// TwinCAT 3 PLC project PLC
// ProgramVersion: 3.1.4024.0
// libraries:
//   EfficientIO Communicator, * (EfficientIO)
//   Lynus Persistent Data V1, * (Lynus AG)
//   Lynus Standards, * (Lynus AG)
//   Tc2_ModbusRTU, * (Beckhoff Automation GmbH)
//   Tc2_SerialCom, * (Beckhoff Automation GmbH)
//   Tc2_Standard, * (Beckhoff Automation GmbH)
//   Tc2_System, * (Beckhoff Automation GmbH)
//   Tc2_Utilities, * (Beckhoff Automation GmbH)
//   Tc3_Module, * (Beckhoff Automation GmbH)
// project tree:
//   DUTs/ ModbusRTURequest.TcDUT
//   / FastTask.TcTTO, MiddleTask.TcTTO, SlowTask.TcTTO
//   FB/ FB_ModBus_2Registers_FC4_T.TcPOU (not stored), F_Convert_Reg_to_Real.TcPOU (not stored), MODBUS_RTU_EcoForest.TcPOU, MODBUS_RTU_Vallox.TcPOU
//   POUs/ prgCom.TcPOU, prgHeatPump.TcPOU, prgMiddle.TcPOU, prgPD.TcPOU, prgRoomVentilaton.TcPOU, prgVar.TcPOU
// real-time tasks:
//   TASK FastTask: cycle T#5ms, priority 19, ADS port 351
//   TASK MiddleTask: cycle T#10ms, priority 20, ADS port 352
//   TASK SlowTask: cycle T#20ms, priority 21, ADS port 353
// I/O:
//   DEVICE Gerät 2 (CX-BK)
//     Box 1 (CX-BK)
// variable links:
//   PLC/PLC Instance <-> Device 2 (CX-BK)/Box 1 (CX-BK)
//     MiddleTask Inputs/MODBUS_RTU_EcoForest.fbModbusRtuMaster_KL6x22B.InData/D[{0..21}] <-> Term 2 (KL6041)/Channel 1/Data In {0..21}  (22 links)
//     MiddleTask Inputs/MODBUS_RTU_EcoForest.fbModbusRtuMaster_KL6x22B.InData/Status <-> Term 2 (KL6041)/Channel 1/Status
//     MiddleTask Inputs/MODBUS_RTU_Vallox.fbModbusRtuMaster_KL6x22B.InData/D[{0..21}] <-> Term 3 (KL6041)/Channel 1/Data In {0..21}  (22 links)
//     MiddleTask Inputs/MODBUS_RTU_Vallox.fbModbusRtuMaster_KL6x22B.InData/Status <-> Term 3 (KL6041)/Channel 1/Status
//     MiddleTask Outputs/MODBUS_RTU_EcoForest.fbModbusRtuMaster_KL6x22B.OutData/Ctrl <-> Term 2 (KL6041)/Channel 1/Ctrl
//     MiddleTask Outputs/MODBUS_RTU_EcoForest.fbModbusRtuMaster_KL6x22B.OutData/D[{0..21}] <-> Term 2 (KL6041)/Channel 1/Data Out {0..21}  (22 links)
//     MiddleTask Outputs/MODBUS_RTU_Vallox.fbModbusRtuMaster_KL6x22B.OutData/Ctrl <-> Term 3 (KL6041)/Channel 1/Ctrl
//     MiddleTask Outputs/MODBUS_RTU_Vallox.fbModbusRtuMaster_KL6x22B.OutData/D[{0..21}] <-> Term 3 (KL6041)/Channel 1/Data Out {0..21}  (22 links)
//     SlowTask Inputs/prgMiddle.uint_State <-> Inputs/State

CONFIGURATION PLC
    RESOURCE PLC ON TwinCAT3
        TASK FastTask(INTERVAL := T#5ms, PRIORITY := 19);
        TASK MiddleTask(INTERVAL := T#10ms, PRIORITY := 20);
        TASK SlowTask(INTERVAL := T#20ms, PRIORITY := 21);
        PROGRAM prgPD WITH FastTask : prgPD;
        PROGRAM prgVar WITH FastTask : prgVar;
        PROGRAM prgMiddle WITH MiddleTask : prgMiddle;
        PROGRAM prgCom WITH SlowTask : prgCom;
    END_RESOURCE
END_CONFIGURATION

// ---- DUTs/ModbusRTURequest.TcDUT
TYPE ModbusRTURequest :
STRUCT
	byteClientSlaveID	:BYTE;
	uintStartAddress	:UINT;
	uintNoOfWords		:UINT;
	mError				:BOOL;
	udintErrorID		:MODBUS_ERRORS;
	udintBytesReceived	:UDINT;
	timerErrorTimer		:TON;
	timerOKTimer		:TON;
	wArrayReceiveBuffer	:ARRAY[0..130] OF WORD;
	udintReceiveBufferAddress	:UDINT;
	strErrorMessage		:STRING(50);
	udintCommErrorCounter		:UDINT;
	udintCommSuccessCounter		:UDINT;
	timeTimeForRequest	:TIME;
	mRequestActive		:BOOL;
	intDeviceClass		:INT;
	intDeviceNumber		:INT;
END_STRUCT
END_TYPE

// ---- POUs/prgPD.TcPOU
PROGRAM prgPD
VAR
	fbPers						: FB_WritePersistentData_General;
	fb_Reboot		: NT_reboot;
	m_Reboot		: BOOL:=FALSE;
END_VAR

fbPers(
	eSaveModeData:= eUSVSaveMode.eSaveEventBased, 
	bLoadPersistentDataOk=> , 
	bError=> , 
	bySaveProcess=> , 
	dwStorageLast24h=> , 
	udiErrorCode=> );
	
	
fb_Reboot(	netid := '',
			delay := 2,
			start := m_Reboot);

END_PROGRAM

// ---- POUs/prgVar.TcPOU
PROGRAM prgVar
VAR
	fbVar			: FB_VarInfo_V3;
	fbrw1			: FB_ReadWrite_V2;
END_VAR

fbVar(
	bReadInfo:= , 
	eTMCFile:= eSelectTMCFile.eDontUseTMCFile, 
	eSavePositionTMCFile:= eSavePositionOnPLC.ePostionHardDisk, 
	udiCounterFoundVariables=> , 
	bError=> , 
	bBusy=> , 
	byProgress=> , 
	udiErrorCodeOut=> , 
	eErrorVarInfo_Out=> , 
	sVarWithError=> );
fbVar();
fbVar();
	
fbRW1(	eUploadType := eSelectDataUploadType.e_Change_Intervall5min,
		bBusy=> , 
		bError=> , 
		udiErrorCodeOut=> , 
		eErrorReadWrite_Out=> );

END_PROGRAM

// ---- POUs/prgMiddle.TcPOU
PROGRAM prgMiddle
VAR
	i: INT;
	int_LiveCount_5min:INT;								//{#lynus.ag#()}
	ton_5min: Ton;
	uint_State								AT%I* 	: UINT;		//{#lynus.ag#()}
	mtest: BOOL;

END_VAR

i:= i+1;
ton_5min( 	In := NOT ton_5min.Q,
			PT := T#5M);
IF ton_5min.Q THEN
	int_LiveCount_5min := int_LiveCount_5min+1;
END_IF

prgHeatPump();
prgRoomVentilaton();

END_PROGRAM

// ---- POUs/prgHeatPump.TcPOU
PROGRAM prgHeatPump
VAR
	fb_word_to_float	:FB_CV_WORD_TO_REAL_FLOAT;
	real_ProductionTemperatureOut		: REAL;									//{#lynus.ag#()}
	real_ProductionTemperatureIn		: REAL;									//{#lynus.ag#()}
	real_CompresorSuctionPressure		: REAL;									//{#lynus.ag#()}
	real_CompressorDischargePressure	: REAL;									//{#lynus.ag#()}
	real_DHWTemperature					: REAL;									//{#lynus.ag#()}
	real_OutdoorTemperature				: REAL;									//{#lynus.ag#()}
	real_BrineCircuitPressure			: REAL;									//{#lynus.ag#()}
	real_ProductionCircuitPressure		: REAL;									//{#lynus.ag#()}
	real_CompressorStartTempForDHW		: REAL;									//{#lynus.ag#()}
	real_COP							: REAL;									//{#lynus.ag#()}
	real_PF								: REAL;									//{#lynus.ag#()}
	real_CondensationTemperature		: REAL;									//{#lynus.ag#()}
	real_Superheat						: REAL;									//{#lynus.ag#()}
	real_ExpansionValvePosition			: REAL;									//{#lynus.ag#()}
	real_SetpointDHWBUS					: REAL;									//{#lynus.ag#()}
	real_BUSHeatingDG1Setpoint			: REAL;									//{#lynus.ag#()}
	real_BUSHeatingSG2Setpoint			: REAL;									//{#lynus.ag#()}
	real_BUSHeatingSG3Setpoint			: REAL;									//{#lynus.ag#()}
	real_BUSHeatingSG4Setpoint			: REAL;									//{#lynus.ag#()}
	real_BUSCoolingDG1Setpoint			: REAL;									//{#lynus.ag#()}
	real_BUSCoolingSG2Setpoint			: REAL;									//{#lynus.ag#()}
	real_BUSCoolingSG3Setpoint			: REAL;									//{#lynus.ag#()}
	real_BUSCoolingSG4Setpoint			: REAL;									//{#lynus.ag#()}
	real_SupplytemperatureSG2			: REAL;									//{#lynus.ag#()}
	real_SupplytemperatureSG3			: REAL;									//{#lynus.ag#()}
	real_SupplytemperatureSG4			: REAL;									//{#lynus.ag#()}
	real_DHWStarttemperature			: REAL;									//{#lynus.ag#()}
	real_Evaporationtemperature			: REAL;									//{#lynus.ag#()}
	real_Heatingbuffertanktemp			: REAL;									//{#lynus.ag#()}
	real_Coolingbuffertanktemp			: REAL;									//{#lynus.ag#()}
	real_EER							: REAL;									//{#lynus.ag#()}
	real_Compresordischargetemp			: REAL;									//{#lynus.ag#()}
	real_Surplusactivationsetpoint		: REAL;									//{#lynus.ag#()}
	real_Consumptionlimitsetpoint 		: REAL;									//{#lynus.ag#()}
	real_CompressorRPM					: REAL;									//{#lynus.ag#()}
	real_ScrollTemp						: REAL;									//{#lynus.ag#()}
	real_Invertertemperature			: REAL;									//{#lynus.ag#()}
	real_Powerconsumption				: REAL;									//{#lynus.ag#()}
	real_Condensationcapacity			: REAL;									//{#lynus.ag#()}

	real_Heatpumpstate					: REAL;									//{#lynus.ag#()}
	// 1=Off; 2=On; 3=Emergency; 0=Keyboard
	real_Workingprogram					: REAL;									//{#lynus.ag#()}
	// 1=Winter;2=Summer; 3=Mixed; 0=Keyboard
	real_BUS_DHWDemand					: REAL;									//{#lynus.ag#()}
	real_BUS_SG2Demand					: REAL;									//{#lynus.ag#()}
	real_BUS_SG3Demand					: REAL;									//{#lynus.ag#()}
	real_BUS_SG4Demand					: REAL;									//{#lynus.ag#()}
//	real_			: REAL;									//{#lynus.ag#()}
//	real_			: REAL;									//{#lynus.ag#()}
	
	bool_HP_Alarm					: BOOL;								//{#lynus.ag#()}
	bool_HP_BusControlEnable		: BOOL;								//{#lynus.ag#()}

	mTest: BOOL;

END_VAR

MODBUS_RTU_EcoForest();
IF MODBUS_RTU_EcoForest.structArrayModbusRTU[1].wArrayReceiveBuffer[10]<>0 THEN 	
	real_ProductionTemperatureOut 	:=INT_TO_REAL(WORD_TO_INT(MODBUS_RTU_EcoForest.structArrayModbusRTU[1].wArrayReceiveBuffer[2]))/10;
	real_ProductionTemperatureIn 	:=INT_TO_REAL(WORD_TO_INT(MODBUS_RTU_EcoForest.structArrayModbusRTU[1].wArrayReceiveBuffer[3]))/10;
	real_CompresorSuctionPressure 	:=INT_TO_REAL(WORD_TO_INT(MODBUS_RTU_EcoForest.structArrayModbusRTU[1].wArrayReceiveBuffer[5]))/10;
	real_CompressorDischargePressure:=int_to_real(word_to_int(MODBUS_RTU_EcoForest.structArrayModbusRTU[1].wArrayReceiveBuffer[6]))/10;
	real_DHWTemperature				:=int_to_real(word_to_int(MODBUS_RTU_EcoForest.structArrayModbusRTU[1].wArrayReceiveBuffer[7]))/10;
	real_OutdoorTemperature			:=int_to_real(word_to_int(MODBUS_RTU_EcoForest.structArrayModbusRTU[1].wArrayReceiveBuffer[10]))/10;
	real_BrineCircuitPressure		:=int_to_real(word_to_int(MODBUS_RTU_EcoForest.structArrayModbusRTU[1].wArrayReceiveBuffer[12]))/10;
	real_ProductionCircuitPressure	:=int_to_real(word_to_int(MODBUS_RTU_EcoForest.structArrayModbusRTU[1].wArrayReceiveBuffer[13]))/10;
	real_CompressorStartTempForDHW	:=int_to_real(word_to_int(MODBUS_RTU_EcoForest.structArrayModbusRTU[1].wArrayReceiveBuffer[14]))/10;
END_IF
IF (MODBUS_RTU_EcoForest.structArrayModbusRTU[2].wArrayReceiveBuffer[7])/10 <> 0 THEN	
	real_COP						:= INT_TO_REAL(WORD_TO_INT(MODBUS_RTU_EcoForest.structArrayModbusRTU[2].wArrayReceiveBuffer[7]))/10;	
	real_PF							:= INT_TO_REAL(WORD_TO_INT(MODBUS_RTU_EcoForest.structArrayModbusRTU[2].wArrayReceiveBuffer[8]))/10;
END_IF	
IF  (MODBUS_RTU_EcoForest.structArrayModbusRTU[3].wArrayReceiveBuffer[0])/10 <>0 THEN 	
	real_CondensationTemperature	:= INT_TO_REAL(WORD_TO_INT(MODBUS_RTU_EcoForest.structArrayModbusRTU[3].wArrayReceiveBuffer[0]))/10;	
END_IF	
IF (MODBUS_RTU_EcoForest.structArrayModbusRTU[4].wArrayReceiveBuffer[1])/10 <> 0 THEN
	real_Superheat					:= INT_TO_REAL(WORD_TO_INT(MODBUS_RTU_EcoForest.structArrayModbusRTU[4].wArrayReceiveBuffer[0]))/10;	
	real_ExpansionValvePosition		:= int_to_real(word_to_int(MODBUS_RTU_EcoForest.structArrayModbusRTU[4].wArrayReceiveBuffer[1]))/10;	
	real_SetpointDHWBUS				:= int_to_real(word_to_int(MODBUS_RTU_EcoForest.structArrayModbusRTU[4].wArrayReceiveBuffer[2]))/10;	
	real_BUSHeatingDG1Setpoint		:= int_to_real(word_to_int(MODBUS_RTU_EcoForest.structArrayModbusRTU[4].wArrayReceiveBuffer[3]))/10;	
	real_BUSHeatingSG2Setpoint		:= int_to_real(word_to_int(MODBUS_RTU_EcoForest.structArrayModbusRTU[4].wArrayReceiveBuffer[4]))/10;	
	real_BUSHeatingSG3Setpoint		:= int_to_real(word_to_int(MODBUS_RTU_EcoForest.structArrayModbusRTU[4].wArrayReceiveBuffer[5]))/10;	
	real_BUSHeatingSG4Setpoint		:= int_to_real(word_to_int(MODBUS_RTU_EcoForest.structArrayModbusRTU[4].wArrayReceiveBuffer[6]))/10;	
	real_BUSCoolingDG1Setpoint		:= int_to_real(word_to_int(MODBUS_RTU_EcoForest.structArrayModbusRTU[4].wArrayReceiveBuffer[7]))/10;	
	real_BUSCoolingSG2Setpoint		:= int_to_real(word_to_int(MODBUS_RTU_EcoForest.structArrayModbusRTU[4].wArrayReceiveBuffer[8]))/10;	
	real_BUSCoolingSG3Setpoint		:= int_to_real(word_to_int(MODBUS_RTU_EcoForest.structArrayModbusRTU[4].wArrayReceiveBuffer[9]))/10;	
	real_BUSCoolingSG4Setpoint		:= INT_TO_REAL(WORD_TO_INT(MODBUS_RTU_EcoForest.structArrayModbusRTU[4].wArrayReceiveBuffer[10]))/10;	
END_IF


IF (MODBUS_RTU_EcoForest.structArrayModbusRTU[7].wArrayReceiveBuffer[1])/10 <> 0 THEN 
	real_SupplytemperatureSG2		:= INT_TO_REAL(WORD_TO_INT(MODBUS_RTU_EcoForest.structArrayModbusRTU[7].wArrayReceiveBuffer[0]))/10;	
	real_SupplytemperatureSG3		:= int_to_real(word_to_int(MODBUS_RTU_EcoForest.structArrayModbusRTU[7].wArrayReceiveBuffer[1]))/10;	
	real_SupplytemperatureSG4		:= int_to_real(word_to_int(MODBUS_RTU_EcoForest.structArrayModbusRTU[7].wArrayReceiveBuffer[2]))/10;	
	real_DHWStarttemperature		:= int_to_real(word_to_int(MODBUS_RTU_EcoForest.structArrayModbusRTU[7].wArrayReceiveBuffer[3]))/10;	
	real_Evaporationtemperature		:= int_to_real(word_to_int(MODBUS_RTU_EcoForest.structArrayModbusRTU[7].wArrayReceiveBuffer[4]))/10;	
	real_Heatingbuffertanktemp		:= int_to_real(word_to_int(MODBUS_RTU_EcoForest.structArrayModbusRTU[7].wArrayReceiveBuffer[5]))/10;	
	real_Coolingbuffertanktemp		:= int_to_real(word_to_int(MODBUS_RTU_EcoForest.structArrayModbusRTU[7].wArrayReceiveBuffer[6]))/10;	
	real_EER						:= int_to_real(word_to_int(MODBUS_RTU_EcoForest.structArrayModbusRTU[7].wArrayReceiveBuffer[7]))/10;	
	real_Compresordischargetemp		:= int_to_real(word_to_int(MODBUS_RTU_EcoForest.structArrayModbusRTU[7].wArrayReceiveBuffer[8]))/10;	
END_IF

IF (MODBUS_RTU_EcoForest.structArrayModbusRTU[8].wArrayReceiveBuffer[0])/10 <> 0 THEN
	real_Surplusactivationsetpoint	:= INT_TO_REAL(WORD_TO_INT(MODBUS_RTU_EcoForest.structArrayModbusRTU[8].wArrayReceiveBuffer[0]))/10;	
	real_Consumptionlimitsetpoint	:= INT_TO_REAL(WORD_TO_INT(MODBUS_RTU_EcoForest.structArrayModbusRTU[8].wArrayReceiveBuffer[1]))/10;	
END_IF

IF MODBUS_RTU_EcoForest.structArrayModbusRTU[5].wArrayReceiveBuffer[3] <> 0 THEN		
	real_CompressorRPM 				:= INT_TO_REAL(WORD_TO_INT(MODBUS_RTU_EcoForest.structArrayModbusRTU[5].wArrayReceiveBuffer[0]));
	real_ScrollTemp					:= int_to_real(word_to_int(MODBUS_RTU_EcoForest.structArrayModbusRTU[5].wArrayReceiveBuffer[2]));
	real_Invertertemperature		:= int_to_real(word_to_int(MODBUS_RTU_EcoForest.structArrayModbusRTU[5].wArrayReceiveBuffer[3]));
END_IF

IF MODBUS_RTU_EcoForest.structArrayModbusRTU[6].wArrayReceiveBuffer[3] <> 0 THEN
	real_Powerconsumption			:= INT_TO_REAL(WORD_TO_INT(MODBUS_RTU_EcoForest.structArrayModbusRTU[6].wArrayReceiveBuffer[2]));		
	real_Condensationcapacity		:= INT_TO_REAL(WORD_TO_INT(MODBUS_RTU_EcoForest.structArrayModbusRTU[6].wArrayReceiveBuffer[3]));		
END_IF

IF MODBUS_RTU_EcoForest.structArrayModbusRTU[9].wArrayReceiveBuffer[8] <> 0 THEN // [8] = Start counter
	real_Heatpumpstate		:= INT_TO_REAL(WORD_TO_INT(MODBUS_RTU_EcoForest.structArrayModbusRTU[9].wArrayReceiveBuffer[0]));	
	real_Workingprogram		:= INT_TO_REAL(WORD_TO_INT(MODBUS_RTU_EcoForest.structArrayModbusRTU[9].wArrayReceiveBuffer[1]));	
	real_BUS_DHWDemand		:= INT_TO_REAL(WORD_TO_INT(MODBUS_RTU_EcoForest.structArrayModbusRTU[9].wArrayReceiveBuffer[2]));
	real_BUS_SG2Demand		:= INT_TO_REAL(WORD_TO_INT(MODBUS_RTU_EcoForest.structArrayModbusRTU[9].wArrayReceiveBuffer[4]));	
	real_BUS_SG3Demand		:= INT_TO_REAL(WORD_TO_INT(MODBUS_RTU_EcoForest.structArrayModbusRTU[9].wArrayReceiveBuffer[5]));	
	real_BUS_SG4Demand		:= INT_TO_REAL(WORD_TO_INT(MODBUS_RTU_EcoForest.structArrayModbusRTU[9].wArrayReceiveBuffer[6]));	
END_IF
	

bool_HP_Alarm 				:= WORD_TO_BOOL(MODBUS_RTU_EcoForest.structArrayModbusRTU[10].wArrayReceiveBuffer[0]);
bool_HP_BusControlEnable	:= WORD_TO_BOOL(MODBUS_RTU_EcoForest.structArrayModbusRTU[10].wArrayReceiveBuffer[3]);

//			:= INT_TO_REAL(WORD_TO_INT(MODBUS_RTU_EcoForest.structArrayModbusRTU[].wArrayReceiveBuffer[]));	
//			:= INT_TO_REAL(WORD_TO_INT(MODBUS_RTU_EcoForest.structArrayModbusRTU[].wArrayReceiveBuffer[]));

END_PROGRAM

// ---- FB/MODBUS_RTU_EcoForest.TcPOU
PROGRAM MODBUS_RTU_EcoForest

VAR_INPUT

END_VAR
VAR_OUTPUT
	dword_MB_Error		:ARRAY[1..3] OF DWORD;
END_VAR
VAR
//	fbModbusRtuMaster_KL6x22B: ModbusRtuMaster_KL6x22B;
	fbModbusRtuMaster_KL6x22B: ModbusRtuMasterV2_KL6x22B;
	fbConfigKL6041 : KL6Configuration;
	uintPollOrderCount: UINT;
	mBusy: BOOL;
	mError: BOOL;
	mStart: BOOL;
	udintMemoryDestAddress: UDINT;
	udintBytesReceived: UDINT;
	intState: INT:=0;
	timerT1: TON;
	timeWaitT1: TIME:=T#500MS;
	timeWaitT2: TIME:=T#500MS;
	timeNoRxTimeout:	TIME:=T#2S;
	timerT2: TON;

	fb_F_TRIG1: F_TRIG;
	timerTimeout: TON;
	mError_Rx: BOOL;
	udintErrorID: MODBUS_ERRORS;
	byteClientSlaveID: BYTE;
	uintNoOfWords: UINT;
	uintStartAddress: UINT;
	dw_Mask: DWORD;
	dw_Mask_Not: DWORD;
	uint_TestPollOrder: UINT;
	mTestMode: BOOL;
	mInit_Done: BOOL;
	
	structArrayModbusRTU	:ARRAY[1..60] OF ModbusRTURequest;
	uintMaxModbusRTUOrders: UINT;
	mExecute: BOOL;
	int_Handshake: ComHandshake_t:=4;
	mode: ComSerialLineMode_t:=3;
	byte_DataBits: BYTE:=8;
	Word_Quantity: WORD;
	Word_Adress: WORD;
	uint_Length: UINT;
	udint_Write_Value:UDINT;
	udintMemoryDestAddress_Write: POINTER TO UDINT;
	mStartWrite: BOOL;
	i:uint;
END_VAR

(*
The function block "ModbusRtuMaster_KL6x22B" has 22 bytes where it communicates with the plc
software. These 22 bytes have to be assigned to the hardware device (for example KL/EL6021) in the
system manager plus the control and status byte.
If devices with less then 22 bytes are used, the other function blocks have to be used (for 5 bytes for example).
*)

(*
IF fbModbusRtuMaster_KL6x22B.MBmaster.TimeoutTON.Q=TRUE AND mTimeOUT_Qold=FALSE THEN mTimeOUT_Q_Rising; END_IF
mTimeOUT_Qold:=fbModbusRtuMaster_KL6x22B.MBmaster.TimeoutTON.Q;
*)

fb_F_TRIG1(CLK:=mBusy);

CASE intState OF

0: 	(* reset the start bit *)
	mStart:=FALSE;
	IF mInit_Done AND NOT fbConfigKL6041.Busy THEN 
		intState:=10;
		mExecute:=FALSE;		
	ELSE
		INIT();
		mExecute:=TRUE;		// necessary to write the communication parameters to the KL terminal. only necessary once if the terminal is brand new
	END_IF
10:
	(* set next poll order *)
	uintPollOrderCount:=uintPollOrderCount+1; (* next slave *)
	WHILE NOT structArrayModbusRTU[uintPollOrderCount].mRequestActive DO
		uintPollOrderCount:=uintPollOrderCount+1; (* next slave *)
	END_WHILE
	
	(* trouble shooting *)
	IF mTestMode THEN
		uintPollOrderCount:=uint_TestPollOrder; (* next slave *)
	END_IF
	
	IF uintPollOrderCount > uintMaxModbusRTUOrders OR uintPollOrderCount<1 THEN
		uintPollOrderCount:=1;
	END_IF

	udintMemoryDestAddress:=ADR(structArrayModbusRTU[uintPollOrderCount].wArrayReceiveBuffer[0]);
	structArrayModbusRTU[uintPollOrderCount].udintBytesReceived:=0;
	mStart:=TRUE;
	timerTimeout.IN:=TRUE;
	intState:=20;

20: (* wait for busy falling or time out *)
	IF fb_F_TRIG1.Q OR timerTimeout.Q THEN

		(* check answer time *)
		structArrayModbusRTU[uintPollOrderCount].timeTimeForRequest:=timerTimeout.ET;

		(* reset timer *)
		timerTimeout.IN:=FALSE;

		(* reset start bit *)
		mStart:=FALSE;

		(* save number of bytes received *)
		structArrayModbusRTU[uintPollOrderCount].udintBytesReceived:=udintBytesReceived;
		udintBytesReceived:=0;

		(* Error Detection *)
		IF timerTimeout.Q THEN
			mError_Rx:=TRUE;
			structArrayModbusRTU[uintPollOrderCount].udintErrorID:=9998;
			structArrayModbusRTU[uintPollOrderCount].strErrorMessage:='Timeout';
		ELSIF structArrayModbusRTU[uintPollOrderCount].udintBytesReceived=0 AND structArrayModbusRTU[uintPollOrderCount].uintNoOfWords>0 THEN
			mError_Rx:=TRUE;
			structArrayModbusRTU[uintPollOrderCount].udintErrorID:=9999;
			structArrayModbusRTU[uintPollOrderCount].strErrorMessage:='0 bytes received';
		ELSIF fbModbusRtuMaster_KL6x22B.Error THEN
			mError_Rx:=TRUE;
			structArrayModbusRTU[uintPollOrderCount].udintErrorID:=udintErrorID;
//			structArrayModbusRTU[uintPollOrderCount].strErrorMessage:=F_ADSERRORTEXT(structArrayModbusRTU[uintPollOrderCount].udintErrorID);
		ELSE
			mError_Rx:=FALSE;
			structArrayModbusRTU[uintPollOrderCount].udintErrorID:=0;
			structArrayModbusRTU[uintPollOrderCount].strErrorMessage:='';
		END_IF


		IF mError_Rx THEN
			structArrayModbusRTU[uintPollOrderCount].udintCommErrorCounter:=structArrayModbusRTU[uintPollOrderCount].udintCommErrorCounter+1;
		ELSIF structArrayModbusRTU[uintPollOrderCount].udintBytesReceived>0 THEN (* Rev 3 *)
			structArrayModbusRTU[uintPollOrderCount].udintCommSuccessCounter:=structArrayModbusRTU[uintPollOrderCount].udintCommSuccessCounter+1;
		END_IF

		structArrayModbusRTU[uintPollOrderCount].timerOKTimer.IN:=NOT mError_Rx;
		structArrayModbusRTU[uintPollOrderCount].timerErrorTimer.IN:=mError_Rx;

		dw_Mask:=1;
		dw_Mask:=SHL(dw_Mask,(structArrayModbusRTU[uintPollOrderCount].intDeviceNumber));
		dw_Mask_Not:=NOT dw_Mask;
		
		IF structArrayModbusRTU[uintPollOrderCount].timerErrorTimer.Q THEN
			structArrayModbusRTU[uintPollOrderCount].mError:=TRUE;
			IF structArrayModbusRTU[uintPollOrderCount].intDeviceClass>=1 AND structArrayModbusRTU[uintPollOrderCount].intDeviceClass<=3 THEN
				dword_MB_Error[structArrayModbusRTU[uintPollOrderCount].intDeviceClass]:=dword_MB_Error[structArrayModbusRTU[uintPollOrderCount].intDeviceClass] OR dw_Mask;
			END_IF
		END_IF

		IF structArrayModbusRTU[uintPollOrderCount].timerOKTimer.Q THEN
			structArrayModbusRTU[uintPollOrderCount].mError:=FALSE;
			IF structArrayModbusRTU[uintPollOrderCount].intDeviceClass>=1 AND structArrayModbusRTU[uintPollOrderCount].intDeviceClass<=3 THEN
				dword_MB_Error[structArrayModbusRTU[uintPollOrderCount].intDeviceClass]:=dword_MB_Error[structArrayModbusRTU[uintPollOrderCount].intDeviceClass] AND dw_Mask_Not;
			END_IF
		END_IF

		(* clear buffer *)
		IF mError_Rx THEN
			MEMSET(destAddr:=udintMemoryDestAddress,fillByte:=0,130);
		END_IF

		(* set next state *)
		intState:=30;
	END_IF

30:		(* wait *)
		timerT1(IN:=TRUE);
		IF timerT1.Q THEN
			timerT1(IN:=FALSE);
			intState:=0; (* back to start *)
		END_IF

END_CASE

(* Timer calls *)
structArrayModbusRTU[uintPollOrderCount].timerErrorTimer(PT:=timeNoRxTimeout);
structArrayModbusRTU[uintPollOrderCount].timerOKTimer(PT:=T#2S);
timerT1(PT:=timeWaitT1);
timerT2(PT:=timeWaitT2);
timerTimeout(PT:=timeNoRxTimeout+timeWaitT1);


(* Timers *)
structArrayModbusRTU[uintPollOrderCount].timerErrorTimer.PT:=T#5S;
structArrayModbusRTU[uintPollOrderCount].timerOKTimer.PT:=T#5S;


//fbModbusRtuMaster_KL6x22B.ReadInputRegs(
fbModbusRtuMaster_KL6x22B.ReadRegs(
	UnitID:= structArrayModbusRTU[uintPollOrderCount].byteClientSlaveID, 
	Quantity:= structArrayModbusRTU[uintPollOrderCount].uintNoOfWords, 
	MBAddr:= structArrayModbusRTU[uintPollOrderCount].uintStartAddress , 
	cbLength:= 2*structArrayModbusRTU[uintPollOrderCount].uintNoOfWords,
	pMemoryAddr:= udintMemoryDestAddress, 
	AuxQuantity:= , 
	AuxMBAddr:= , 
	AuxcbLength:= , 
	pAuxMemoryAddr:= , 
	Execute:= mStart, 
	Timeout:= T#1S, 
	BUSY=> mBusy, 
	Error=> mError, 
	ErrorId=> udintErrorID, 
	cbRead=> udintBytesReceived);
	
(*fbModbusRtuMaster_KL6x22B.ReadRegs(
	UnitID		:=structArrayModbusRTU[uintPollOrderCount].byteClientSlaveID,
	Quantity	:=structArrayModbusRTU[uintPollOrderCount].uintNoOfWords,
	MBAddr		:=structArrayModbusRTU[uintPollOrderCount].uintStartAddress,
	cbLength	:=2*structArrayModbusRTU[uintPollOrderCount].uintNoOfWords,
	pMemoryAddr	:=udintMemoryDestAddress,
	Execute		:=mStart,
	Timeout		:=t#1s,
	BUSY		=>mBusy,
	Error		=>mError,
	ErrorId		=>udintErrorID,
	cbRead		=>udintBytesReceived
);
*)
(*
(*fbModbusRtuMaster_KL6x22B.ReadInputRegs(
*)
fbModbusRtuMaster_KL6x22B.ReadInputRegs(
	UnitID		:=structArrayModbusRTU[uintPollOrderCount].byteClientSlaveID,
	Quantity	:=structArrayModbusRTU[uintPollOrderCount].uintNoOfWords,
	MBAddr		:=structArrayModbusRTU[uintPollOrderCount].uintStartAddress,
	cbLength	:=2*structArrayModbusRTU[uintPollOrderCount].uintNoOfWords,
	pMemoryAddr	:=udintMemoryDestAddress,
	Execute		:=mStart,
	Timeout		:=t#1s,
	BUSY		=>mBusy,
	Error		=>mError,
	ErrorId		=>udintErrorID,
	cbRead		=>udintBytesReceived
);
*)
// necessary for KL6041 to wirte the com settings
fbConfigKL6041(
	Execute 		:= mExecute,
	Mode 			:= mode,
	Baudrate 		:= 19200,
	NoDatabits 		:= byte_DataBits,
	Parity 			:= 0,
	Stopbits 		:= 2,
	Handshake  		:= int_Handshake,
	ContinousMode 	:= FALSE,
	pComIn 			:= ADR(fbModbusRtuMaster_KL6x22B.InData),
	pComOut 		:= ADR(fbModbusRtuMaster_KL6x22B.OutData),
	SizeComIn 		:= SIZEOF(fbModbusRtuMaster_KL6x22B.InData)
);

fbModbusRtuMaster_KL6x22B.WriteRegs(
	UnitID:= structArrayModbusRTU[uintPollOrderCount].byteClientSlaveID, 
	AuxQuantity:= Word_Quantity, 
	AuxMBAddr:= Word_Adress, 
	AuxcbLength:= uint_Length,
	pAuxMemoryAddr:= udintMemoryDestAddress_Write, 
	Execute:= mStartWrite, 
	Timeout:= T#1S, 
	BUSY=> mBusy, 
	Error=> mError, 
	ErrorId=> udintErrorID, 
	cbRead=> udintBytesReceived);

udintMemoryDestAddress_Write:=ADR(udint_Write_Value);

ACTION INIT:
(* Poll 1 *)
i:=1;
structArrayModbusRTU[i].byteClientSlaveID:=17;
structArrayModbusRTU[i].uintStartAddress:=1;
structArrayModbusRTU[i].uintNoOfWords:=22;
structArrayModbusRTU[i].mRequestActive:=TRUE;
                     
(* Poll 2 *)  
i:=i+1;       
structArrayModbusRTU[i].byteClientSlaveID:=17;
structArrayModbusRTU[i].uintStartAddress:=23;
structArrayModbusRTU[i].uintNoOfWords:=22;
structArrayModbusRTU[i].mRequestActive:=TRUE;
                     
(* Poll 3 *)  
i:=i+1;       
structArrayModbusRTU[i].byteClientSlaveID:=17;
structArrayModbusRTU[i].uintStartAddress:=94;
structArrayModbusRTU[i].uintNoOfWords:=1;
structArrayModbusRTU[i].mRequestActive:=TRUE;
                     
(* Poll 4 *) 
i:=i+1;        
structArrayModbusRTU[i].byteClientSlaveID:=17;
structArrayModbusRTU[i].uintStartAddress:=132;
structArrayModbusRTU[i].uintNoOfWords:=22;
structArrayModbusRTU[i].mRequestActive:=TRUE;
                
(* Poll 5 *) 
i:=i+1;        
structArrayModbusRTU[i].byteClientSlaveID:=17;
structArrayModbusRTU[i].uintStartAddress:=5002;
structArrayModbusRTU[i].uintNoOfWords:=6;
structArrayModbusRTU[i].mRequestActive:=TRUE;
                     
(* Poll 6 *) 
i:=i+1;        
structArrayModbusRTU[i].byteClientSlaveID:=17;
structArrayModbusRTU[i].uintStartAddress:=5080;
structArrayModbusRTU[i].uintNoOfWords:=22;
structArrayModbusRTU[i].mRequestActive:=TRUE;

(* Poll 7 *) 
i:=i+1;        
structArrayModbusRTU[i].byteClientSlaveID:=17;
structArrayModbusRTU[i].uintStartAddress:=194;
structArrayModbusRTU[i].uintNoOfWords:=22;
structArrayModbusRTU[i].mRequestActive:=TRUE;

(* Poll 8 *) 
i:=i+1;        
structArrayModbusRTU[i].byteClientSlaveID:=17;
structArrayModbusRTU[i].uintStartAddress:=2000;
structArrayModbusRTU[i].uintNoOfWords:=2;
structArrayModbusRTU[i].mRequestActive:=TRUE;

(* Poll 9 *) 
i:=i+1;        
structArrayModbusRTU[i].byteClientSlaveID:=17;
structArrayModbusRTU[i].uintStartAddress:=5220;
structArrayModbusRTU[i].uintNoOfWords:=22;
structArrayModbusRTU[i].mRequestActive:=TRUE;

(* Poll 10 *) 
i:=i+1;        
structArrayModbusRTU[i].byteClientSlaveID:=17;
structArrayModbusRTU[i].uintStartAddress:=50;
structArrayModbusRTU[i].uintNoOfWords:=4;
structArrayModbusRTU[i].mRequestActive:=TRUE;




uintMaxModbusRTUOrders:=i;
mInit_Done:=TRUE;
END_ACTION

END_PROGRAM

// ---- POUs/prgRoomVentilaton.TcPOU
PROGRAM prgRoomVentilaton
VAR
	real_Ventialtor_Speed		: REAL;									//{#lynus.ag#()}
	real_Temp_Extract_Air		: REAL;									//{#lynus.ag#()}
	real_Temp_Exhaust_Air		: REAL;									//{#lynus.ag#()}
	real_Temp_Outdoor_Air		: REAL;									//{#lynus.ag#()}
	real_Temp_Supply_Cell_Air	: REAL;									//{#lynus.ag#()}
	real_Temp_Supply_Air		: REAL;									//{#lynus.ag#()}
	real_Humidity				: REAL;									//{#lynus.ag#()}
	real_CO2					: REAL;									//{#lynus.ag#()}
	
END_VAR

MODBUS_RTU_Vallox();
IF (WORD_TO_REAL(MODBUS_RTU_Vallox.structArrayModbusRTU[1].wArrayReceiveBuffer[3])-27315)/100 <> 0 AND (WORD_TO_REAL(MODBUS_RTU_Vallox.structArrayModbusRTU[1].wArrayReceiveBuffer[10]))/1 <> 0 THEN 
	real_Ventialtor_Speed := WORD_TO_REAL(MODBUS_RTU_Vallox.structArrayModbusRTU[1].wArrayReceiveBuffer[0]);
	real_Temp_Extract_Air := (WORD_TO_REAL(MODBUS_RTU_Vallox.structArrayModbusRTU[1].wArrayReceiveBuffer[1])-27315)/100;
	real_Temp_Exhaust_Air := (WORD_TO_REAL(MODBUS_RTU_Vallox.structArrayModbusRTU[1].wArrayReceiveBuffer[2])-27315)/100;
	real_Temp_Outdoor_Air := (WORD_TO_REAL(MODBUS_RTU_Vallox.structArrayModbusRTU[1].wArrayReceiveBuffer[3])-27315)/100;
	real_Temp_Supply_Cell_Air := (WORD_TO_REAL(MODBUS_RTU_Vallox.structArrayModbusRTU[1].wArrayReceiveBuffer[4])-27315)/100;
	real_Temp_Supply_Air := (WORD_TO_REAL(MODBUS_RTU_Vallox.structArrayModbusRTU[1].wArrayReceiveBuffer[5])-27315)/100;
	real_Humidity		 := (WORD_TO_REAL(MODBUS_RTU_Vallox.structArrayModbusRTU[1].wArrayReceiveBuffer[10]))/1;
	real_CO2			 := (WORD_TO_REAL(MODBUS_RTU_Vallox.structArrayModbusRTU[1].wArrayReceiveBuffer[11]))/1;
END_IF

END_PROGRAM

// ---- FB/MODBUS_RTU_Vallox.TcPOU
PROGRAM MODBUS_RTU_Vallox

VAR_INPUT

END_VAR
VAR_OUTPUT
	dword_MB_Error		:ARRAY[1..3] OF DWORD;
END_VAR
VAR
//	fbModbusRtuMaster_KL6x22B: ModbusRtuMaster_KL6x22B;
	fbModbusRtuMaster_KL6x22B: ModbusRtuMasterV2_KL6x22B;
	fbConfigKL6041 : KL6Configuration;
	uintPollOrderCount: UINT;
	mBusy: BOOL;
	mError: BOOL;
	mStart: BOOL;
	udintMemoryDestAddress: UDINT;
	udintBytesReceived: UDINT;
	intState: INT:=0;
	timerT1: TON;
	timeWaitT1: TIME:=T#500MS;
	timeWaitT2: TIME:=T#500MS;
	timeNoRxTimeout:	TIME:=T#2S;
	timerT2: TON;

	fb_F_TRIG1: F_TRIG;
	timerTimeout: TON;
	mError_Rx: BOOL;
	udintErrorID: MODBUS_ERRORS;
	byteClientSlaveID: BYTE;
	uintNoOfWords: UINT;
	uintStartAddress: UINT;
	dw_Mask: DWORD;
	dw_Mask_Not: DWORD;
	uint_TestPollOrder: UINT;
	mTestMode: BOOL;
	mInit_Done: BOOL;
	
	structArrayModbusRTU	:ARRAY[1..60] OF ModbusRTURequest;
	uintMaxModbusRTUOrders: UINT;
	mExecute: BOOL;
	int_Handshake: ComHandshake_t:=4;
	mode: ComSerialLineMode_t:=3;
	byte_DataBits: BYTE:=8;
END_VAR

(*
The function block "ModbusRtuMaster_KL6x22B" has 22 bytes where it communicates with the plc
software. These 22 bytes have to be assigned to the hardware device (for example KL/EL6021) in the
system manager plus the control and status byte.
If devices with less then 22 bytes are used, the other function blocks have to be used (for 5 bytes for example).
*)

(*
IF fbModbusRtuMaster_KL6x22B.MBmaster.TimeoutTON.Q=TRUE AND mTimeOUT_Qold=FALSE THEN mTimeOUT_Q_Rising; END_IF
mTimeOUT_Qold:=fbModbusRtuMaster_KL6x22B.MBmaster.TimeoutTON.Q;
*)

fb_F_TRIG1(CLK:=mBusy);

CASE intState OF

0: 	(* reset the start bit *)
	mStart:=FALSE;
	IF mInit_Done AND NOT fbConfigKL6041.Busy THEN 
		intState:=10;
		mExecute:=FALSE;		
	ELSE
		INIT();
		mExecute:=TRUE;		// necessary to write the communication parameters to the KL terminal. only necessary once if the terminal is brand new
	END_IF
10:
	(* set next poll order *)
	uintPollOrderCount:=uintPollOrderCount+1; (* next slave *)
	WHILE NOT structArrayModbusRTU[uintPollOrderCount].mRequestActive DO
		uintPollOrderCount:=uintPollOrderCount+1; (* next slave *)
	END_WHILE
	
	(* trouble shooting *)
	IF mTestMode THEN
		uintPollOrderCount:=uint_TestPollOrder; (* next slave *)
	END_IF
	
	IF uintPollOrderCount > uintMaxModbusRTUOrders OR uintPollOrderCount<1 THEN
		uintPollOrderCount:=1;
	END_IF

	udintMemoryDestAddress:=ADR(structArrayModbusRTU[uintPollOrderCount].wArrayReceiveBuffer[0]);
	structArrayModbusRTU[uintPollOrderCount].udintBytesReceived:=0;
	mStart:=TRUE;
	timerTimeout.IN:=TRUE;
	intState:=20;

20: (* wait for busy falling or time out *)
	IF fb_F_TRIG1.Q OR timerTimeout.Q THEN

		(* check answer time *)
		structArrayModbusRTU[uintPollOrderCount].timeTimeForRequest:=timerTimeout.ET;

		(* reset timer *)
		timerTimeout.IN:=FALSE;

		(* reset start bit *)
		mStart:=FALSE;

		(* save number of bytes received *)
		structArrayModbusRTU[uintPollOrderCount].udintBytesReceived:=udintBytesReceived;
		udintBytesReceived:=0;

		(* Error Detection *)
		IF timerTimeout.Q THEN
			mError_Rx:=TRUE;
			structArrayModbusRTU[uintPollOrderCount].udintErrorID:=9998;
			structArrayModbusRTU[uintPollOrderCount].strErrorMessage:='Timeout';
		ELSIF structArrayModbusRTU[uintPollOrderCount].udintBytesReceived=0 AND structArrayModbusRTU[uintPollOrderCount].uintNoOfWords>0 THEN
			mError_Rx:=TRUE;
			structArrayModbusRTU[uintPollOrderCount].udintErrorID:=9999;
			structArrayModbusRTU[uintPollOrderCount].strErrorMessage:='0 bytes received';
		ELSIF fbModbusRtuMaster_KL6x22B.Error THEN
			mError_Rx:=TRUE;
			structArrayModbusRTU[uintPollOrderCount].udintErrorID:=udintErrorID;
//			structArrayModbusRTU[uintPollOrderCount].strErrorMessage:=F_ADSERRORTEXT(structArrayModbusRTU[uintPollOrderCount].udintErrorID);
		ELSE
			mError_Rx:=FALSE;
			structArrayModbusRTU[uintPollOrderCount].udintErrorID:=0;
			structArrayModbusRTU[uintPollOrderCount].strErrorMessage:='';
		END_IF


		IF mError_Rx THEN
			structArrayModbusRTU[uintPollOrderCount].udintCommErrorCounter:=structArrayModbusRTU[uintPollOrderCount].udintCommErrorCounter+1;
		ELSIF structArrayModbusRTU[uintPollOrderCount].udintBytesReceived>0 THEN (* Rev 3 *)
			structArrayModbusRTU[uintPollOrderCount].udintCommSuccessCounter:=structArrayModbusRTU[uintPollOrderCount].udintCommSuccessCounter+1;
		END_IF

		structArrayModbusRTU[uintPollOrderCount].timerOKTimer.IN:=NOT mError_Rx;
		structArrayModbusRTU[uintPollOrderCount].timerErrorTimer.IN:=mError_Rx;

		dw_Mask:=1;
		dw_Mask:=SHL(dw_Mask,(structArrayModbusRTU[uintPollOrderCount].intDeviceNumber));
		dw_Mask_Not:=NOT dw_Mask;
		
		IF structArrayModbusRTU[uintPollOrderCount].timerErrorTimer.Q THEN
			structArrayModbusRTU[uintPollOrderCount].mError:=TRUE;
			IF structArrayModbusRTU[uintPollOrderCount].intDeviceClass>=1 AND structArrayModbusRTU[uintPollOrderCount].intDeviceClass<=3 THEN
				dword_MB_Error[structArrayModbusRTU[uintPollOrderCount].intDeviceClass]:=dword_MB_Error[structArrayModbusRTU[uintPollOrderCount].intDeviceClass] OR dw_Mask;
			END_IF
		END_IF

		IF structArrayModbusRTU[uintPollOrderCount].timerOKTimer.Q THEN
			structArrayModbusRTU[uintPollOrderCount].mError:=FALSE;
			IF structArrayModbusRTU[uintPollOrderCount].intDeviceClass>=1 AND structArrayModbusRTU[uintPollOrderCount].intDeviceClass<=3 THEN
				dword_MB_Error[structArrayModbusRTU[uintPollOrderCount].intDeviceClass]:=dword_MB_Error[structArrayModbusRTU[uintPollOrderCount].intDeviceClass] AND dw_Mask_Not;
			END_IF
		END_IF

		(* clear buffer *)
		IF mError_Rx THEN
			MEMSET(destAddr:=udintMemoryDestAddress,fillByte:=0,130);
		END_IF

		(* set next state *)
		intState:=30;
	END_IF

30:		(* wait *)
		timerT1(IN:=TRUE);
		IF timerT1.Q THEN
			timerT1(IN:=FALSE);
			intState:=0; (* back to start *)
		END_IF

END_CASE

(* Timer calls *)
structArrayModbusRTU[uintPollOrderCount].timerErrorTimer(PT:=timeNoRxTimeout);
structArrayModbusRTU[uintPollOrderCount].timerOKTimer(PT:=T#2S);
timerT1(PT:=timeWaitT1);
timerT2(PT:=timeWaitT2);
timerTimeout(PT:=timeNoRxTimeout+timeWaitT1);


(* Timers *)
structArrayModbusRTU[uintPollOrderCount].timerErrorTimer.PT:=T#5S;
structArrayModbusRTU[uintPollOrderCount].timerOKTimer.PT:=T#5S;


//fbModbusRtuMaster_KL6x22B.ReadInputRegs(
fbModbusRtuMaster_KL6x22B.ReadRegs(
	UnitID:= structArrayModbusRTU[uintPollOrderCount].byteClientSlaveID, 
	Quantity:= structArrayModbusRTU[uintPollOrderCount].uintNoOfWords, 
	MBAddr:= structArrayModbusRTU[uintPollOrderCount].uintStartAddress , 
	cbLength:= 2*structArrayModbusRTU[uintPollOrderCount].uintNoOfWords,
	pMemoryAddr:= udintMemoryDestAddress, 
	AuxQuantity:= , 
	AuxMBAddr:= , 
	AuxcbLength:= , 
	pAuxMemoryAddr:= , 
	Execute:= mStart, 
	Timeout:= T#1S, 
	BUSY=> mBusy, 
	Error=> mError, 
	ErrorId=> udintErrorID, 
	cbRead=> udintBytesReceived);
	
(*fbModbusRtuMaster_KL6x22B.ReadRegs(
	UnitID		:=structArrayModbusRTU[uintPollOrderCount].byteClientSlaveID,
	Quantity	:=structArrayModbusRTU[uintPollOrderCount].uintNoOfWords,
	MBAddr		:=structArrayModbusRTU[uintPollOrderCount].uintStartAddress,
	cbLength	:=2*structArrayModbusRTU[uintPollOrderCount].uintNoOfWords,
	pMemoryAddr	:=udintMemoryDestAddress,
	Execute		:=mStart,
	Timeout		:=t#1s,
	BUSY		=>mBusy,
	Error		=>mError,
	ErrorId		=>udintErrorID,
	cbRead		=>udintBytesReceived
);
*)
(*
(*fbModbusRtuMaster_KL6x22B.ReadInputRegs(
*)
fbModbusRtuMaster_KL6x22B.ReadInputRegs(
	UnitID		:=structArrayModbusRTU[uintPollOrderCount].byteClientSlaveID,
	Quantity	:=structArrayModbusRTU[uintPollOrderCount].uintNoOfWords,
	MBAddr		:=structArrayModbusRTU[uintPollOrderCount].uintStartAddress,
	cbLength	:=2*structArrayModbusRTU[uintPollOrderCount].uintNoOfWords,
	pMemoryAddr	:=udintMemoryDestAddress,
	Execute		:=mStart,
	Timeout		:=t#1s,
	BUSY		=>mBusy,
	Error		=>mError,
	ErrorId		=>udintErrorID,
	cbRead		=>udintBytesReceived
);
*)
// necessary for KL6041 to wirte the com settings
fbConfigKL6041(
	Execute 		:= mExecute,
	Mode 			:= mode,
	Baudrate 		:= 19200,
	NoDatabits 		:= byte_DataBits,
	Parity 			:= 1,
	Stopbits 		:= 1,
	Handshake  		:= int_Handshake,
	ContinousMode 	:= FALSE,
	pComIn 			:= ADR(fbModbusRtuMaster_KL6x22B.InData),
	pComOut 		:= ADR(fbModbusRtuMaster_KL6x22B.OutData),
	SizeComIn 		:= SIZEOF(fbModbusRtuMaster_KL6x22B.InData)
);

ACTION INIT:



(* Poll 1 Heating circuit 1 *)
structArrayModbusRTU[1].byteClientSlaveID:=1;
structArrayModbusRTU[1].uintStartAddress:=4353;
structArrayModbusRTU[1].uintNoOfWords:=22;
structArrayModbusRTU[1].mRequestActive:=TRUE;


uintMaxModbusRTUOrders:=1;
mInit_Done:=TRUE;
END_ACTION

END_PROGRAM

// ---- POUs/prgCom.TcPOU
PROGRAM prgCom
VAR
	fbCom			: FB_MqttCommunicator_V3;
END_VAR

fbCom(
	bConnect:= TRUE, 
	strAuthKey					:=  'TSG88376368072' ,
	sUserName:= '2ba1290e-1bda-4738-b4d7-c3a5a574d522', 
	sUserPassword:= 'ce0e73e8-643a-4866-98c1-79497096b888', 
	eSavePositionCertificate:= eSavePositionOnPLC.ePostionHardDisk,
	bConnected=> , 
	bError=> , 
	hrErrorCode=> , 
	eConnectionState=> , 
	eErrorMessage_Out=> );

END_PROGRAM
